FUNCTION_BLOCK FB_Machine
VAR_INPUT
END_VAR
VAR_OUTPUT
END_VAR
VAR
	//Buttons
	Start		: ST_LEDButton;
	HMI_Start	: ST_LEDButton;
	rtStart		: R_TRIG;
	Stop		: ST_LEDButton;
	HMI_Stop	: ST_LEDButton;
	rtStop		: R_TRIG;
	Reset		: ST_LEDButton;
	HMI_Reset	: ST_LEDButton;
	rtReset		: R_TRIG;

	//Inputs
	LocalEstop AT %I*	: BOOL;
	MachineAIn			: ST_MachineModuleInputs;
	MachineBIn			: ST_MachineModuleInputs;
	MachineCIn			: ST_MachineModuleInputs;
	MachineDIn			: ST_MachineModuleInputs;

	//Overide
	Override : LREAL := 30.0;

	TwinSAFEGroupRun			AT %Q*	: BOOL := TRUE;
	TwinSAFEGroupErrAck			AT %Q*	: BOOL;
	TwinSAFEGroupState			AT %I*	: USINT;
	TwinSAFE_X_Axis_ActPos		AT %Q*	: UDINT;
	TwinSAFE_ResetAllEstopZones	AT %Q*	: BOOL;

	TwinSAFE_Machine_A_Estop_State	AT %I*	: USINT;
	TwinSAFE_Machine_B_Estop_State	AT %I*	: USINT;
	TwinSAFE_Machine_C_Estop_State	AT %I*	: USINT;
	TwinSAFE_Machine_D_Estop_State	AT %I*	: USINT;

	AxisInError : BOOL; //One or more axis in error

	X_Axis			: AXIS_REF;
	Z_Axis			: AXIS_REF;
	fbCarrierReset	: FB_CarrierReset;

	fbCarrierStop : FB_CarrierStop;

	StateToReturnToAfterStop	: E_State;
	lastState					: E_State;
	previousState				: E_State;
	State						: E_State;
	NextState					: E_State;

	//HMI Display               		
	sPreviouseState : STRING;

	sState : STRING;

	sNextState : STRING;

	fbMoveCarrier		: FB_CarrierAbsMove;
	HomePosSetPoint		: ST_CarrierSetPoint	:= (X_Pos := 100, X_Velo := 500, Z_Pos := 100, Z_Velo := 800);
	APickPosSetPoint	: ST_CarrierSetPoint	:= (X_Pos := 290, X_Velo := 500, Z_Pos := 1100, Z_Velo := 800);
	BWaitPosSetpoint	: ST_CarrierSetPoint	:= (X_Pos := 600, X_Velo := 500, Z_Pos := 100, Z_Velo := 800);
	BPlacePosSetPoint	: ST_CarrierSetPoint	:= (X_Pos := 1000, X_Velo := 500, Z_Pos := 1200, Z_Velo := 800);
	BWorkPosSetPoint	: ST_CarrierSetPoint	:= (X_Pos := 1000, X_Velo := 500, Z_Pos := 100, Z_Velo := 800);
	BPickPosSetPoint	: ST_CarrierSetPoint	:= (X_Pos := 1000, X_Velo := 500, Z_Pos := 1200, Z_Velo := 800);
	CWaitPosSetPoint	: ST_CarrierSetPoint	:= (X_Pos := 1350, X_Velo := 500, Z_Pos := 100, Z_Velo := 800);
	CPlacePosSetPoint	: ST_CarrierSetPoint	:= (X_Pos := 1700, X_Velo := 500, Z_Pos := 1000, Z_Velo := 800);
	CWorkPosSetPoint	: ST_CarrierSetPoint	:= (X_Pos := 1800, X_Velo := 500, Z_Pos := 100, Z_Velo := 800);

	//Machine A                 		
	WaitTimeForAToBeReady : TIME := T#1S;

	//Machine B             		
	WaitTimeForBtoBeReady	: TIME	:= T#1.5S;
	BDoingWorkTime			: TIME	:= T#2S;

	//Machine C             			
	WaitTimeForCtoBeReady	: TIME	:= T#0.5S;
	CDoingWorkTime			: TIME	:= T#750MS;

	//Machine D
	Machine_D_Carrier_Gripper AT %Q* : BIT;

	//Event Logger - Clear messages on reset
	//fbEventLogger : FB_TcEventLogger;

	iResetingStep : UDINT;

	//Alarms
	//Drive not ready error
	X_AxisDriveNotReady	: FB_AlarmWrapper;
	Z_AxisDriveNotReady	: FB_AlarmWrapper;

	//Catch all axis error      		
	X_AxisError	: FB_AlarmWrapper;
	Z_AxisError	: FB_AlarmWrapper;

	//one of the Estop buttons is pressed
	AlarmLocalEstopPressed		: FB_AlarmWrapper;
	AlarmMachineAEstopPressed	: FB_AlarmWrapper;
	AlarmMachineBEstopPressed	: FB_AlarmWrapper;
	AlarmMachineCEstopPressed	: FB_AlarmWrapper;
	AlarmMachineDEstopPressed	: FB_AlarmWrapper;

	//one of the light curtains is tripped
	AlarmMachineALightCurtain	: FB_AlarmWrapper;
	AlarmMachineBLightCurtain	: FB_AlarmWrapper;
	AlarmMachineCLightCurtain	: FB_AlarmWrapper;

	//The TwinSAFE E-Stop fuction block is tripped
	AlarmMachineAEstopTripped	: FB_AlarmWrapper;
	AlarmMachineBEstopTripped	: FB_AlarmWrapper;
	AlarmMachineCEstopTripped	: FB_AlarmWrapper;
	AlarmMachineDEstopTripped	: FB_AlarmWrapper;
END_VAR



rtStart(CLK := Start.Button OR HMI_Start.Button);
rtStop(CLK := Stop.Button OR HMI_Stop.Button);
rtReset(CLK := Reset.Button OR HMI_Reset.Button);

M_HMI_Display();

CASE State OF
	E_State.Init:
		fbMoveCarrier.X_AxisRef	:= ADR(X_Axis);
		fbMoveCarrier.Z_AxisRef	:= ADR(Z_Axis);
		fbMoveCarrier(Execute := FALSE);
		Machine_D_Carrier_Gripper := FALSE;

		fbCarrierReset(Execute := FALSE);
		fbCarrierReset.X_AxisRef	:= ADR(X_Axis);
		fbCarrierReset.Z_AxisRef	:= ADR(Z_Axis);

		fbCarrierStop(Execute := FALSE);
		fbCarrierStop.X_AxisRef	:= ADR(X_Axis);
		fbCarrierStop.Z_AxisRef	:= ADR(Z_Axis);

		State			:= E_State.Idel;
		NextState		:= E_State.Idel;
		iResetingStep	:= 0;
	E_State.Idel:
		NextState := E_State.Enable;

		IF TwinSAFEGroupState = 1 AND NOT AxisInError THEN
			IF rtStart.Q THEN
				State := E_State.Enable;
			ELSIF rtReset.Q THEN
				State := E_State.Reseting;
			ELSIF AxisInError THEN
				State := E_State.Error;
			END_IF
		ELSE
			State := E_State.Error;
		END_IF

	E_State.Enable:
		NextState := E_State.MoveToHome;

		IF TwinSAFEGroupState = 1 THEN
			State := E_State.MoveToHome;
		ELSIF AxisInError OR TwinSAFEGroupState <> 1 THEN
			State := E_State.Error;
		END_IF

	E_State.MoveToHome:
		NextState					:= E_State.WaitForAToBeReady;
		StateToReturnToAfterStop	:= State;
		fbMoveCarrier.SetPoint		:= HomePosSetPoint;
		fbMoveCarrier(Execute := TRUE);

		IF fbMoveCarrier.Done THEN
			fbMoveCarrier(Execute := FALSE);
			State := E_State.WaitForAToBeReady;
		ELSIF fbMoveCarrier.Error THEN
			State := E_State.Error;
		END_IF

	E_State.WaitForAToBeReady:
		NextState					:= E_State.MoveToAPickPos;
		StateToReturnToAfterStop	:= State;

		IF M_ProcessDelay(WaitTimeForAToBeReady) THEN
			State := E_State.MoveToAPickPos;
		END_IF

	E_State.MoveToAPickPos:
		NextState					:= E_State.PickFromA;
		StateToReturnToAfterStop	:= State;
		fbMoveCarrier.SetPoint		:= APickPosSetPoint;
		fbMoveCarrier(Execute := TRUE);

		IF fbMoveCarrier.Done THEN
			fbMoveCarrier(Execute := FALSE);
			State := E_State.PickFromA;
		ELSIF fbMoveCarrier.Error THEN
			State := E_State.Error;
		END_IF

	E_State.PickFromA:
		NextState					:= E_State.MoveToBWaitPos;
		StateToReturnToAfterStop	:= State;

		IF M_CloseGripper() THEN
			State := E_State.MoveToBWaitPos;
		END_IF

	E_State.MoveToBWaitPos:
		NextState					:= E_State.WaitForBToBeReady;
		StateToReturnToAfterStop	:= State;
		fbMoveCarrier.SetPoint		:= BWaitPosSetpoint;
		fbMoveCarrier(Execute := TRUE);

		IF fbMoveCarrier.Done THEN
			fbMoveCarrier(Execute := FALSE);
			State := E_State.WaitForBToBeReady;
		ELSIF fbMoveCarrier.Error THEN
			State := E_State.Error;
		END_IF

	E_State.WaitForBToBeReady:
		NextState					:= E_State.MoveToBPlacePosition;
		StateToReturnToAfterStop	:= State;

		IF M_ProcessDelay(WaitTimeForBtoBeReady) THEN
			State := E_State.MoveToBPlacePosition;
		END_IF

	E_State.MoveToBPlacePosition:
		NextState					:= E_State.PlaceOnB;
		StateToReturnToAfterStop	:= State;
		fbMoveCarrier.SetPoint		:= BPlacePosSetPoint;
		fbMoveCarrier(Execute := TRUE);

		IF fbMoveCarrier.Done THEN
			fbMoveCarrier(Execute := FALSE);
			State := E_State.PlaceOnB;
		ELSIF fbMoveCarrier.Error THEN
			State := E_State.Error;
		END_IF

	E_State.PlaceOnB:
		NextState					:= E_State.MoveToBWorkPos;
		StateToReturnToAfterStop	:= State;

		IF M_OpenGripper() THEN
			State := E_State.MoveToBWorkPos;
		END_IF

	E_State.MoveToBWorkPos:
		NextState					:= E_State.BDoingWork;
		StateToReturnToAfterStop	:= State;
		fbMoveCarrier.SetPoint		:= BWorkPosSetPoint;
		fbMoveCarrier(Execute := TRUE);

		IF fbMoveCarrier.Done THEN
			fbMoveCarrier(Execute := FALSE);
			State := E_State.BDoingWork;
		ELSIF fbMoveCarrier.Error THEN
			State := E_State.Error;
		END_IF

	E_State.BDoingWork:
		NextState					:= E_State.MoveToBPickPos;
		StateToReturnToAfterStop	:= State;

		IF M_ProcessDelay(BDoingWorkTime) THEN
			State := E_State.MoveToBPickPos;
		END_IF

	E_State.MoveToBPickPos:
		NextState					:= E_State.PickPartFromB;
		StateToReturnToAfterStop	:= State;
		fbMoveCarrier.SetPoint		:= BPickPosSetPoint;
		fbMoveCarrier(Execute := TRUE);

		IF fbMoveCarrier.Done THEN
			fbMoveCarrier(Execute := FALSE);
			State := E_State.PickPartFromB;
		ELSIF fbMoveCarrier.Error THEN
			State := E_State.Error;
		END_IF

	E_State.PickPartFromB:
		NextState					:= E_State.MoveToCWaitPos;
		StateToReturnToAfterStop	:= State;

		IF M_CloseGripper() THEN
			State := E_State.MoveToCWaitPos;
		END_IF

	E_State.MoveToCWaitPos:
		NextState					:= E_State.WaitForCToBeReady;
		StateToReturnToAfterStop	:= State;
		fbMoveCarrier.SetPoint		:= CWaitPosSetPoint;
		fbMoveCarrier(Execute := TRUE);

		IF fbMoveCarrier.Done THEN
			fbMoveCarrier(Execute := FALSE);
			State := E_State.WaitForCToBeReady;
		ELSIF fbMoveCarrier.Error THEN
			State := E_State.Error;
		END_IF

	E_State.WaitForCToBeReady:
		NextState					:= E_State.MoveToCPlacePos;
		StateToReturnToAfterStop	:= State;

		IF M_ProcessDelay(WaitTimeForCtoBeReady) THEN
			State := E_State.MoveToCPlacePos;
		END_IF

	E_State.MoveToCPlacePos:
		NextState					:= E_State.PlaceOnC;
		StateToReturnToAfterStop	:= State;
		fbMoveCarrier.SetPoint		:= CPlacePosSetPoint;
		fbMoveCarrier(Execute := TRUE);

		IF fbMoveCarrier.Done THEN
			fbMoveCarrier(Execute := FALSE);
			State := E_State.PlaceOnC;
		ELSIF fbMoveCarrier.Error THEN
			State := E_State.Error;
		END_IF

	E_State.PlaceOnC:
		NextState					:= E_State.MoveToCWorkPos;
		StateToReturnToAfterStop	:= State;

		IF M_OpenGripper() THEN
			State := E_State.MoveToCWorkPos;
		END_IF

	E_State.MoveToCWorkPos:
		NextState					:= E_State.CDoingWork;
		StateToReturnToAfterStop	:= State;
		fbMoveCarrier.SetPoint		:= CWorkPosSetPoint;
		fbMoveCarrier(Execute := TRUE);

		IF fbMoveCarrier.Done THEN
			fbMoveCarrier(Execute := FALSE);
			State := E_State.CDoingWork;
		ELSIF fbMoveCarrier.Error THEN
			State := E_State.Error;
		END_IF

	E_State.CDoingWork:
		NextState					:= E_State.MoveToHome;
		StateToReturnToAfterStop	:= State;

		IF M_ProcessDelay(CDoingWorkTime) THEN
			State := E_State.MoveToHome;
		END_IF

	E_State.Stopping:
		NextState := E_State.Stopped;
		fbCarrierStop(Execute := TRUE);

		IF fbCarrierStop.Done THEN
			fbCarrierStop(Execute := FALSE);
			State := E_State.Stopped;
		ELSIF fbCarrierStop.Error THEN
			State := E_State.Error;
		END_IF

	E_State.Stopped:
		NextState := StateToReturnToAfterStop;

		IF rtStart.Q THEN
			fbMoveCarrier(Execute := FALSE);
			State := StateToReturnToAfterStop;
		END_IF

	E_State.Error:
		NextState := E_State.Reseting;

		IF rtReset.Q THEN
			State := E_State.Reseting;
		END_IF

	E_State.Reseting:
		NextState := E_State.Init;

		CASE iResetingStep OF
			0: //Clear out event logger
				//IF fbEventLogger.ClearLoggedEvents(0) THEN
				iResetingStep := 10;
			//END_IF

			10: //Toggle TS group Err ack
				TwinSAFEGroupErrAck	:= TRUE;
				iResetingStep		:= 20;

			20: //Clear axis error
				fbCarrierReset(Execute := TRUE);
				TwinSAFEGroupErrAck := FALSE;

				IF NOT fbCarrierReset.Busy THEN
					fbCarrierReset(Execute := FALSE);
					State := E_State.Init;
				END_IF
		END_CASE

END_CASE

M_AxisPower();
M_Alarms();
M_BtnLights();
M_ToTwinSAFE();

METHOD M_Alarms
VAR_INPUT
END_VAR
VAR_INST

	InitStep	: UDINT	:= 0;
	initDone	: BOOL	:= FALSE;

	fbReadXAxis	: MC_ReadParameterSet;
	XParams		: ST_AxisParameterSet;
	fbReadZAxis	: MC_ReadParameterSet;
	ZParams		: ST_AxisParameterSet;
END_VAR
IF NOT initDone THEN
	CASE InitStep OF
		0: //Create events
			X_AxisError.Create(stEventEntry := TC_EVENTS.DriveErrors.AxisInError);
			Z_AxisError.Create(stEventEntry := TC_EVENTS.DriveErrors.AxisInError);

			X_AxisDriveNotReady.Create(stEventEntry := TC_EVENTS.DriveErrors.DriveHardwareNotReadyToOperate);
			Z_AxisDriveNotReady.Create(stEventEntry := TC_EVENTS.DriveErrors.DriveHardwareNotReadyToOperate);

			AlarmLocalEstopPressed.Create(stEventEntry := TC_EVENTS.SafetyApplication.EstopBtnPressed);
			AlarmMachineAEstopPressed.Create(stEventEntry := TC_EVENTS.SafetyApplication.EstopBtnPressed);
			AlarmMachineBEstopPressed.Create(stEventEntry := TC_EVENTS.SafetyApplication.EstopBtnPressed);
			AlarmMachineCEstopPressed.Create(stEventEntry := TC_EVENTS.SafetyApplication.EstopBtnPressed);
			AlarmMachineDEstopPressed.Create(stEventEntry := TC_EVENTS.SafetyApplication.EstopBtnPressed);

			AlarmMachineALightCurtain.Create(stEventEntry := TC_EVENTS.SafetyApplication.LightCurtainTripped);
			AlarmMachineBLightCurtain.Create(stEventEntry := TC_EVENTS.SafetyApplication.LightCurtainTripped);
			AlarmMachineCLightCurtain.Create(stEventEntry := TC_EVENTS.SafetyApplication.LightCurtainTripped);

			AlarmMachineAEstopTripped.Create(stEventEntry := TC_EVENTS.SafetyApplication.MachineXEstopTripped);
			AlarmMachineBEstopTripped.Create(stEventEntry := TC_EVENTS.SafetyApplication.MachineXEstopTripped);
			AlarmMachineCEstopTripped.Create(stEventEntry := TC_EVENTS.SafetyApplication.MachineXEstopTripped);
			AlarmMachineDEstopTripped.Create(stEventEntry := TC_EVENTS.SafetyApplication.MachineXEstopTripped);

			InitStep := 10;

		10: //Get data for arguments
			fbReadXAxis(Parameter := XParams,
						Axis	:= X_Axis,
						Execute := TRUE);

			fbReadZAxis(Parameter := ZParams,
						Axis	:= Z_Axis,
						Execute := TRUE);

			IF NOT fbReadXAxis.Busy AND NOT fbReadZAxis.Busy THEN
				InitStep := 20;
			END_IF

		20:
			AlarmLocalEstopPressed.Arg0 := 'Local';

			AlarmMachineAEstopPressed.Arg0	:= 'A';
			AlarmMachineBEstopPressed.Arg0	:= 'B';
			AlarmMachineCEstopPressed.Arg0	:= 'C';
			AlarmMachineDEstopPressed.Arg0	:= 'D';

			AlarmMachineALightCurtain.Arg0	:= 'A';
			AlarmMachineBLightCurtain.Arg0	:= 'B';
			AlarmMachineCLightCurtain.Arg0	:= 'C';

			AlarmMachineAEstopTripped.Arg0	:= 'A';
			AlarmMachineBEstopTripped.Arg0	:= 'B';
			AlarmMachineCEstopTripped.Arg0	:= 'C';
			AlarmMachineDEstopTripped.Arg0	:= 'D';

			X_AxisDriveNotReady.Arg0	:= XParams.sAxisName;
			X_AxisError.Arg0			:= XParams.sAxisName;

			Z_AxisDriveNotReady.Arg0	:= ZParams.sAxisName;
			Z_AxisError.Arg0			:= ZParams.sAxisName;

			InitStep	:= 30;
			initDone	:= TRUE;
	END_CASE

	RETURN;
END_IF

//Trigger events

//Estop buttons
AlarmLocalEstopPressed.Cyclic(AlarmState := LocalEstop);

AlarmMachineAEstopPressed.Cyclic(AlarmState := NOT MachineAIn.EstopBtn);
AlarmMachineBEstopPressed.Cyclic(AlarmState := NOT MachineBIn.EstopBtn);
AlarmMachineCEstopPressed.Cyclic(AlarmState := NOT MachineCIn.EstopBtn);
AlarmMachineDEstopPressed.Cyclic(AlarmState := NOT MachineDIn.EstopBtn);

AlarmMachineALightCurtain.Cyclic(AlarmState := NOT MachineAIn.LightCurtain);
AlarmMachineBLightCurtain.Cyclic(AlarmState := NOT MachineBIn.LightCurtain);
AlarmMachineCLightCurtain.Cyclic(AlarmState := NOT MachineCIn.LightCurtain);

//TwinSAFE logic
AlarmMachineAEstopTripped.Cyclic(AlarmState := TwinSAFE_Machine_A_Estop_State > 1);
AlarmMachineBEstopTripped.Cyclic(AlarmState := TwinSAFE_Machine_B_Estop_State > 1);
AlarmMachineCEstopTripped.Cyclic(AlarmState := TwinSAFE_Machine_C_Estop_State > 1);
AlarmMachineDEstopTripped.Cyclic(AlarmState := TwinSAFE_Machine_D_Estop_State > 1);

//Axis
X_AxisDriveNotReady.Cyclic(AlarmState := X_Axis.Status.ErrorID = 16#4650);
X_AxisError.Arg1 := TO_STRING(X_Axis.Status.ErrorID);
X_AxisError.Cyclic(AlarmState := X_Axis.Status.ErrorID <> 0 AND X_Axis.Status.ErrorID <> 16#4650);

Z_AxisDriveNotReady.Cyclic(AlarmState := Z_Axis.Status.ErrorID = 16#4650);
Z_AxisError.Arg1 := TO_STRING(Z_Axis.Status.ErrorID);
Z_AxisError.Cyclic(AlarmState := Z_Axis.Status.ErrorID <> 0 AND Z_Axis.Status.ErrorID <> 16#4650);
END_METHOD

METHOD M_AxisPower : BOOL
VAR_INPUT
END_VAR
VAR_INST
	X_Power	: MC_Power;
	Z_Power	: MC_Power;
END_VAR
X_Power(Axis			:= X_Axis,
		Enable			:= TRUE,
		Enable_Positive := TRUE,
		Enable_Negative := TRUE,
		Override		:= Override);

Z_Power(Axis			:= Z_Axis,
		Enable			:= TRUE,
		Enable_Positive := TRUE,
		Enable_Negative := TRUE,
		Override		:= Override);

X_Axis.ReadStatus();
Z_Axis.ReadStatus();

AxisInError := X_Axis.Status.Error OR Z_Axis.Status.Error;
END_METHOD

METHOD M_BtnLights
VAR_INPUT
END_VAR
VAR_INST					
	StartLEDBlink	: BLINK;
	ResetLEDBlink	: BLINK;
	StopLEDBlink	: BLINK;
END_VAR
//Buttons
//Start
CASE State OF
	E_State.Init:
		Start.LED := FALSE;
	E_State.Idel:
		StartLEDBlink.TIMEHIGH	:= T#1S;
		StartLEDBlink.TIMELOW	:= T#1S;
		Start.LED				:= StartLEDBlink.out;
	E_State.Enable:
		StartLEDBlink.TIMEHIGH	:= T#500MS;
		StartLEDBlink.TIMELOW	:= T#500MS;
		Start.LED				:= StartLEDBlink.out;
	E_State.MoveToHome..E_State.CDoingWork:
		Start.LED := TRUE;
	E_State.Stopping:
		Start.LED := FALSE;
	E_State.Stopped:
		StartLEDBlink.TIMEHIGH	:= T#200MS;
		StartLEDBlink.TIMELOW	:= T#200MS;
		Start.LED				:= StartLEDBlink.out;
	E_State.Error..E_State.Reseting:
		Start.LED := FALSE;
END_CASE

HMI_Start.LED := Start.LED;
StartLEDBlink(ENABLE := TRUE);

//Reset
CASE State OF
	E_State.Init..E_State.CDoingWork:
		Reset.LED := FALSE;
	E_State.Error:
		ResetLEDBlink.TIMEHIGH	:= T#1S;
		ResetLEDBlink.TIMELOW	:= T#1S;
		Reset.LED				:= ResetLEDBlink.OUT;
	E_State.Reseting:
		ResetLEDBlink.TIMEHIGH	:= T#500MS;
		ResetLEDBlink.TIMELOW	:= T#500MS;
		Reset.LED				:= ResetLEDBlink.OUT;
END_CASE

HMI_Reset.LED := Reset.LED;
ResetLEDBlink(ENABLE := TRUE);

//Stop
CASE State OF
	E_State.Init..E_State.Enable:
		Stop.LED := FALSE;
	E_State.MoveToHome..E_State.CDoingWork:
		IF rtStop.Q THEN
			State := E_State.Stopping;
		END_IF

		Stop.LED := TRUE;
	E_State.Stopping:
		StopLEDBlink.TIMEHIGH	:= T#500MS;
		StopLEDBlink.TIMELOW	:= T#500MS;
		Stop.LED				:= StopLEDBlink.OUT;
	E_State.Stopped..E_State.Reseting:
		Stop.LED := FALSE;
END_CASE

HMI_Stop.LED := Stop.LED;
StopLEDBlink(ENABLE := TRUE);
END_METHOD

METHOD M_CloseGripper : BOOL
VAR_INPUT
END_VAR

VAR_INST
	tonDelay : TON;
END_VAR
tonDelay(IN := TRUE, PT := T#200MS);

Machine_D_Carrier_Gripper := TRUE;

IF tonDelay.Q THEN
	tonDelay(IN := FALSE);
	M_CloseGripper := TRUE;
END_IF
END_METHOD

METHOD M_HMI_Display
VAR_INPUT
END_VAR
(* Check if state has changed since the last cycle *)
IF lastState <> State THEN
	previousState := lastState; (* Update previous state *)
END_IF;

(* Update lastState for the next cycle *)
lastState := State;

//HMI Display strings
sPreviouseState	:= F_E_State_To_String(previousState);
sState			:= F_E_State_To_String(State);
sNextState		:= F_E_State_To_String(NextState);
END_METHOD

METHOD M_OpenGripper : BOOL
VAR_INPUT
END_VAR
VAR_INST
	tonDelay : TON;
END_VAR
tonDelay(IN := TRUE, PT := T#200MS);
Machine_D_Carrier_Gripper := FALSE;

IF tonDelay.Q THEN
	tonDelay(IN := FALSE);
	M_OpenGripper := TRUE;
END_IF
END_METHOD

METHOD M_ProcessDelay : BOOL
VAR_INPUT
	pt : TIME;
END_VAR
VAR_INST
	tonDelay : TON;
END_VAR
tonDelay(IN := TRUE, PT := pt, Q =>, ET =>);

IF tonDelay.Q THEN
	M_ProcessDelay := TRUE;
	tonDelay(IN := FALSE, PT := pt, Q =>, ET =>);
END_IF
END_METHOD

METHOD M_ToTwinSAFE
VAR_INPUT
END_VAR
TwinSAFE_X_Axis_ActPos := TO_UDINT(X_Axis.NcToPlc.ActPos);

TwinSAFE_ResetAllEstopZones := Reset.Button OR HMI_Reset.Button;


TwinSAFEGroupRun := TRUE;
END_METHOD

END_FUNCTION_BLOCK

(* stored: Version 1.1.0.1, ProductVersion 3.1.4024.13
   POU FB_Machine: Id {b7e2ee06-f24d-46a5-a5b3-e60b99cad5e4}, SpecialFunc None
   Method M_Alarms: Id {0d27ec4f-fbc2-4610-bb3d-2907967d60dc}
   Method M_AxisPower: Id {677ce463-30f2-4570-893a-c6b140cbb6b7}
   Method M_BtnLights: Id {af046070-a77a-47ce-80e9-2f5b081ed094}
   Method M_CloseGripper: Id {bb5f6fbc-361e-4823-9fe0-7bae5c45e5a8}
   Method M_HMI_Display: Id {2b28b642-ef01-438d-ac1c-6fcbb9133807}
   Method M_OpenGripper: Id {bc5ae333-e81c-4a39-98d0-d42ee8d75e01}
   Method M_ProcessDelay: Id {3395a5bb-7516-43c6-b5c3-a43eefaec935}
   Method M_ToTwinSAFE: Id {cf48c3d9-39ce-4201-a195-96504adf0d58} *)
